RoboDK station: RoboDkSetup_FinalVersion.rdk

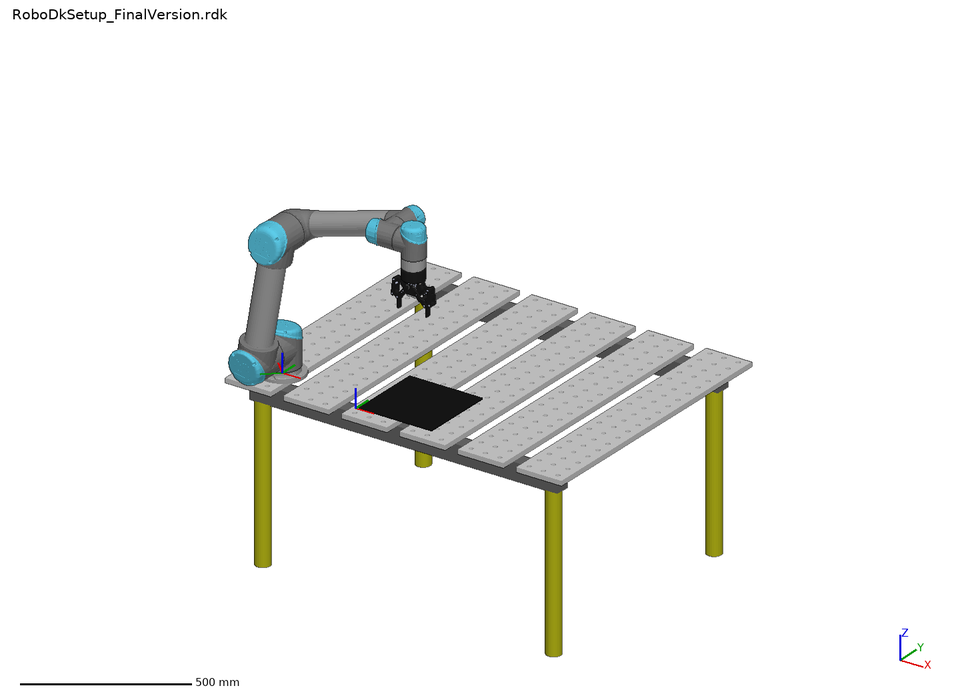
[picture v0: the station drawn from its stored meshes, robots at their saved joint values, targets as dots, program paths as lines]
Station RoboDkSetup_FinalVersion (saved by RoboDK 5.4.1). Poses are relative to the parent item; angles as X-Y-Z fixed-axis rotations.
  - frame UR5 Base at (0, 0, 0) mm, rotated rx 0 ry 0 rz 135.5 deg
    - robot UR5: 6 axes, payload 5 kg, reach 850 mm, repeatability 0.1 mm, weight 18.4 kg
        modified DH rows (alpha deg, a mm, theta deg, d mm): 0, 0, 0, 89.2; 90, 0, 180, 0; 0, 425, 0, 0; 0, 392.43, 0, 109; -90, 0, 0, 93.65; 90, 0, 180, 82
        joint limits [-360, -360, -360, -360, -360, -360] to [360, 360, 360, 360, 360, 360]; home [0, -90, -90, 0, 90, 0]; saved at [-135.592, -99.76, -64.057, -106.183, -270, -87.536]
      - tool GripperA, TCP at (0, 0, 145) mm, size 147.4 x 146.8 x 75 mm
  - frame World at (0, 0, 0) mm
    - object Table at (480, 360, 0) mm, size 1193.8 x 965.2 x 609.6 mm, geometry from welding_table.sld
      - object kameraholder_v2 at (540, -30, 540) mm, rotated rx -90 ry 0 rz 90 deg, size 50 x 40 x 49 mm, geometry from kameraholder_v2.STL
        - object stang_holder at (10, 0, 30) mm, rotated rx -90 ry 0 rz 0 deg, size 29 x 29 x 40 mm, geometry from stang_holder.STL
      - object strueplade at (500, 20, 0) mm, rotated rx 90 ry 0 rz 0 deg, size 50 x 40 x 50 mm, geometry from strueplade.STL
        - object stang_holder at (10, 40, 10) mm, rotated rx 90 ry 0 rz 0 deg, size 29 x 29 x 40 mm, geometry from stang_holder.STL
          - object alu_profil at (5, 5, 0) mm, rotated rx -90 ry 0 rz 0 deg, size 20 x 496 x 20 mm, geometry from alu_profil.STL
  - frame Part1 at (309.75, -70, 0) mm
    - object Plate_Pick at (270, 0, 0) mm, size 260 x 260 x 5 mm, geometry from Plate.step
  - Python program CornerTest (listed below)
  - Python program PickOneBrick (listed below)
  - Python program PickOneFigure (listed below)

--- Python program CornerTest ---
from robolink import *    # API to communicate with RoboDK
from robodk import *      # basic matrix operations
from random import uniform
import numpy as np

# Link to RoboDK
RDK = Robolink()

# define default approach distance
APPROACH = 100

# gather robot from the station
robot               = RDK.Item('UR5', ITEM_TYPE_ROBOT)

# Define the 4 corners of the A3 paper used for the vision
Location = np.array([[0,0,0],
 [283, 0, 0],
 [283, 402, 0],
 [0, 402, 0]])



# ---------------------------------------------------------------------------------
# -------------------------- PROGRAM START ----------------------------------------
#A while loop is set up where it steps on the differet lines in the locations array. So for every time it goes through the loop it goes to a new line.
i = 0
while i <= 3:
    #Here it creats a target of hwere the corner are.
    target_i = transl(Location[i])*rotx(pi)
    #here it creats a targe for approaching the corner so it moves vertical down
    target_i_app = target_i * transl(0,0,-(APPROACH))
    #Moves to th approach location
    robot.MoveL(target_i_app)
    #Moves to the location
    robot.MoveL(target_i)
    #Takes a break on 5 seconds, to see if the grippers are in the right spot
    robot.Pause(5000)
    #Moves the robot back up
    robot.MoveL(target_i_app)
    #adds 1 to the variable of the while loop
    i=i+1

--- Python program PickOneBrick ---
from robolink import *    # API to communicate with RoboDK
from robodk import *      # basic matrix operations
from random import uniform
import numpy as np

# Link to RoboDK
RDK = Robolink()

# define default approach distance
APPROACH = 100

# gather robot from the station
robot               = RDK.Item('UR5', ITEM_TYPE_ROBOT)

#Create an array with the 1 row and 5 columns filled with zeroes
Location = np.zeros(shape=(1,5))

#Reads the csv file, where it sees first splits it in to the different rows
with open('C:/Users/bette/OneDrive/Skrivebord/Final_program/Location.csv', newline= '\n') as csvfile:
    #Here it starts a loop for that are running for all the lines there are in the csv file
    for line in csvfile:
        #splitting the rows up in different columns by the ","
        elements = line[0:-2].split(',')
        #The first column is an index so therefor the x coordinat will be the second column in the csv file, and there for the 1
        x = float(elements[1])
        #Define the 2 column as the y coordinate from the csv file
        y = float(elements[2])
        #Define the 3 column as the z coordinate from the csv file
        z = float(elements[3])
        #Define the 4 column as the rot from the csv file
        rot = float(elements[4])
        #Define the 5 column as the figur number from the csv file
        figur = float(elements[5])
        #adding the new row to the Location array by using the np.vstack.
        Location = np.vstack((Location,[x,y,z,rot,figur]))

#Because of the zero line created at the start and the first row being and index row the first row is deleted twice
Location = np.delete(Location, 0, 0)
Location = np.delete(Location, 0, 0)

#setting up and array with the location of the placement. Here it steps on the z coordinate every new row, and for every third it steps on the y coordinate
Place = np.array([[-100,0,0,0],
                 [-100,0,16,0],
                 [-100,0,32,0],
                 [-100,50,0,0],
                 [-100,50,16,0],
                 [-100,50,32,0],
                 [-100,100,0,0],
                 [-100,100,16,0],
                 [-100,100,32,0],
                 [-100,150,0,0],
                 [-100,150,16, 0],
                 [-100,150,32,0],
                 [-100,200,0,0],
                 [-100,200,16,0],
                 [-100,200,32,0]])

#setting up an definition, that steps on the variable k and the Location array
def MoveBrick(k,Location):
    #create a target of the first row in the loation array
    target_i = transl(Location[0])*rotx(pi)*rotz(2*pi/360*Location[0,3]-(0.25*pi))
    #create a approach target 10 cm over the location
    target_i_app = target_i * transl(0,0,-(APPROACH))
    #moves to the approach location
    robot.MoveL(target_i_app)
    #Moves vertical down to the brick
    robot.MoveL(target_i)
    #takes a pause of 0.5 second
    robot.Pause(500)
    #Next two lines closes the grippers
    robot.setDO(0,0)
    robot.setDO(1,1)
    #takes a pause of 0.5 second
    robot.Pause(500)
    #moves to the approach location
    robot.MoveL(target_i_app)
    #Setting up the placement location by looking at the Place array, and the variable k
    target_i2 = transl(Place[k])*rotx(pi)*rotz(2*pi/360*Place[k,3])
    #creating a approach for the placement
    target_i_app2 = target_i2 * transl(0,0,-(APPROACH))
    #moves to the approach placement
    robot.MoveL(target_i_app2)
    #Moves to the placement
    robot.MoveL(target_i2)
    #takes a pause of 0.5 second
    robot.Pause(500)
    #opening the grippers
    robot.setDO(0,1)
    robot.setDO(1,0)
    #takes a pause of 0.5 second
    robot.Pause(500)
    #moves to the approach placement
    robot.MoveL(target_i_app2)


# ---------------------------------------------------------------------------------
# -------------------------- PROGRAM START ----------------------------------------
#setting up variable i which are used in the while loop
i = 1
#Setting up varianle k, which are used to call the correct placement location
k=0
#Starting the while loop that steps on the varibale i until it gets bigger than 5
while i <= 5:
    #checking if the i is equal to the last column in the first row of the location array.
    if i == Location[0,4]:
        #calling the MoveBrick difinition
        MoveBrick(k,Location)
        #deleting the first location in the array as it is now used
        Location = np.delete(Location, 0, 0)
        #adding 1 to the variable k because of the placement loction now being used.
        k=k+1
        #checking if the i is equal to the last column in the 1 row of the location array
        if i == Location[0,4]:
            #calling the MoveBrick difinition
            MoveBrick(k,Location)
            #deleting the first location in the array as it is now used
            Location = np.delete(Location, 0, 0)
            #adding 1 to the variable k because of the placement loction now being used.
            k=k+1
            #checking if the i is equal to the last column in the 1 row of the location array. If this was maggie being created this will be the only time this will be pass
            if i == Location[0,4]:
                #calling the MoveBrick difinition
                MoveBrick(k,Location)
                #deleting the first location in the array as it is now used
                Location = np.delete(Location, 0, 0)
                #adding 1 to the variable k because of the placement loction now being used.
                k=k+1
            pass
        pass
    pass
    #add 1 to i
    i=i+1

--- Python program PickOneFigure ---
from robolink import *    # API to communicate with RoboDK
from robodk import *      # basic matrix operations
from random import uniform
import numpy as np

# Link to RoboDK
RDK = Robolink()

# define default approach distance
APPROACH = 100

# gather robot from the station
robot               = RDK.Item('UR5', ITEM_TYPE_ROBOT)

Location = np.zeros(shape=(1,5))

with open('C:/Users/bette/OneDrive/Skrivebord/Final_program/Location.csv', newline= '\n') as csvfile:
    for line in csvfile:
        elements = line[0:-2].split(',')
        x = float(elements[1])
        y = float(elements[2])
        z = float(elements[3])
        rot = float(elements[4])
        figur = float(elements[5])
        Location = np.vstack((Location,[x,y,z,rot,figur]))

Location = np.delete(Location, 0, 0)
Location = np.delete(Location, 0, 0)


print(Location)

Place = np.array([[-100,0,40,0],
                 [-100,-30,40,0],
                 [20,-60,40,0],
                 [30,-90,40,0],
                 [40,-120,20,0]])


# ---------------------------------------------------------------------------------
# -------------------------- PROGRAM START ----------------------------------------
i = 1
while i <= 5:
    if i == Location[0,4]:
        target_i = transl(Location[0])*rotx(pi)*rotz(2*pi/360*Location[0,3]-(0.25*pi))
        target_i_app = target_i * transl(0,0,-(APPROACH))
        robot.MoveL(target_i_app)
        robot.MoveL(target_i)
        robot.setDO(0,0)
        robot.setDO(1,1)
        robot.Pause(1000)
        robot.MoveL(target_i_app)
        Location = np.delete(Location, 0, 0)
        if i == Location[0,4]:
            target_i = transl(Location[0])*rotx(pi)*rotz(2*pi/360*Location[0,3]-(0.25*pi))
            target_i_app = target_i * transl(0,0,-(APPROACH))
            robot.MoveL(target_i_app)
            robot.MoveL(target_i)
            robot.Pause(1000)
            robot.MoveL(target_i_app)
            Location = np.delete(Location, 0, 0)
            if i == Location[0,4]:
                target_i = transl(Location[0])*rotx(pi)*rotz(2*pi/360*Location[0,3]-(0.25*pi))
                target_i_app = target_i * transl(0,0,-(APPROACH))
                robot.MoveL(target_i_app)
                robot.MoveL(target_i)
                robot.Pause(1000)
                robot.MoveL(target_i_app)
                Location = np.delete(Location, 0, 0)
            pass
        pass
        target_i2 = transl(Place[i-1])*rotx(pi)*rotz(2*pi/360*Place[i-1,3])
        target_i_app2 = target_i2 * transl(0,0,-(APPROACH))
        robot.MoveL(target_i_app2)
        robot.MoveL(target_i2)
        robot.setDO(0,1)
        robot.setDO(1,0)
        robot.Pause(1000)
        robot.MoveL(target_i_app2)
    pass
    i=i+1
